KUKA KRL program: vw_mod_usr_r.src, vw_mod_usr_r.dat

--- vw_mod_usr_r.src ---
&ACCESS RV2
&REL 1
&COMMENT KS26
&PARAM TPUSER_VERSION = 8.3.0
&PARAM DISKPATH = KRC:\R1\VW_User\Applikation\Projekt_Modul
DEF VW_MOD_USR_R( )
;
;***************************************************
;*Technologiepaket Projekt Modul                   *
;*                                                 *
;*Konzernstandard                                  *
;*Bearbeiter: C. Eisenknappl AUDI AG I/PG-C61      *
;*                                                 *
;* Erstellt am:                                    *
;*                                                 *
;***************************************************
;
END
;
;FOLD MOD1_Interface
GLOBAL DEF MOD1_Interface(USER_CMD:IN,CMD_SEL:IN,PAR1:IN,PAR2:IN,PAR3:IN,PAR4:IN,PAR5:IN,PAR6:IN,PAR7:IN,PAR8:IN,PAR9:IN)
DECL VW_USER_CMD USER_CMD
INT  CMD_SEL,PAR1,PAR2,PAR3,PAR4,PAR5,PAR6,PAR7,PAR8,PAR9
INT i
BOOL bRet
;
SWITCH USER_CMD
;
;***************************************************
  CASE #USR_INIT
    ;FOLD Init
    ;
    ;
    ;ENDFOLD (Init)
;
;***************************************************
  CASE #USR_ADV
    ;FOLD Advance
    ;
    ;
    ;ENDFOLD (Advance)
;
;***************************************************
  CASE #USR_TRIG
    ;FOLD Trig
    ;
    ;
    ;ENDFOLD (TRIG)
;
;***************************************************
  CASE #USR_MAIN
    ;FOLD Main
    ;
    ;
    ;ENDFOLD (Main)
;
;***************************************************
  CASE #USR_MAKRO
    ;FOLD MAKRO
    ;
    ;
    ;ENDFOLD (Makro)
    ;
;***************************************************
ENDSWITCH ;(USER_CMD)
END
;
;ENDFOLD (MOD1_Interface)
;
;***************************************************
;FOLD MOD1 Zangenfunktion
;
;
;ENDFOLD (Zangenfunktion)
;
;***************************************************
;FOLD MOD1_Meldungen
DEF MOD1_Msg(msg_nr :IN, MsgTyp :IN)
INT msg_nr
DECL MOD1R_MsgType MsgTyp
DECL KrlMsg_T USER_MSG
DECL KrlMsgPar_T Par[3]
DECL KrlMsgOpt_T Opt
DECL STATE_T Stat
;
USER_MSG={ Modul[] "MOD1_R_Msg", Nr -1, Msg_txt[] " "}
Opt={ VL_Stop TRUE, Clear_P_Reset TRUE, Log_To_DB FALSE }
Par[1]={ Par_type #Value, Par_txt[] " " }
;
IF ((n_MOD1R_Handle[msg_nr]<0) OR (MsgTyp==#NotifyMsg) OR (MsgTyp==#QuitMsg)) THEN
  USER_MSG.Nr=msg_nr
  SWITCH msg_nr
    CASE 1
      USER_MSG.MSG_TXT[]=" "
    CASE 2
      USER_MSG.MSG_TXT[]=" "
    CASE 3
      USER_MSG.MSG_TXT[]=" "
    CASE 4
      USER_MSG.MSG_TXT[]=" "
    CASE 5
      USER_MSG.MSG_TXT[]=" "
    CASE 6
      USER_MSG.MSG_TXT[]=" "
    CASE 7
      USER_MSG.MSG_TXT[]=" "
    CASE 8
      USER_MSG.MSG_TXT[]=" "
    CASE 9
      USER_MSG.MSG_TXT[]=" "
    CASE 10
      USER_MSG.MSG_TXT[]=" "
    DEFAULT
      USER_MSG.MSG_TXT[]="unbekannte Meldung"
  ENDSWITCH
  SWITCH MsgTyp
    CASE #StateMsg
      n_MOD1R_Handle[msg_nr]=Set_KrlMsg (#State, USER_MSG, Par[], Opt) ;Ausgabe Statusmeldung
    CASE #QuitMsg
      n_MOD1R_Handle[msg_nr]=Set_KrlMsg (#Quit, USER_MSG, Par[], Opt) ;Ausgabe Quittierungsmeldung
      WHILE (Exists_KrlMsg(n_MOD1R_Handle[msg_nr]))  ;Warten bis der Anwender quittiert
        WAIT SEC 0.1
      ENDWHILE
    CASE #NotifyMsg
      n_MOD1R_Handle[msg_nr]=Set_KrlMsg (#Notify, USER_MSG, Par[], Opt) ;Ausgabe Hinweismeldung
    DEFAULT
      n_MOD1R_Handle[msg_nr]=Set_KrlMsg (#Quit, USER_MSG, Par[], Opt) ;Ausgabe Quittierungsmeldung
  ENDSWITCH
ENDIF
END
;
;ENDFOLD (MOD1 Meldungen)
;
;***************************************************
;FOLD MOD2_Interface
GLOBAL DEF MOD2_Interface(USER_CMD:IN,CMD_SEL:IN,PAR1:IN,PAR2:IN,PAR3:IN,PAR4:IN,PAR5:IN,PAR6:IN,PAR7:IN,PAR8:IN,PAR9:IN)
DECL VW_USER_CMD USER_CMD
INT  CMD_SEL,PAR1,PAR2,PAR3,PAR4,PAR5,PAR6,PAR7,PAR8,PAR9
INT i
BOOL bRet
;
SWITCH USER_CMD
;
;***************************************************
  CASE #USR_INIT
    ;FOLD Init
    ;
    $OUT[O_BT_FEHL] = FALSE
    $FLAG[F_X_Lauf_nio] = FALSE
    $FLAG[F_Y_Lauf_nio] = FALSE
    $FLAG[F_Z_Lauf_nio] = FALSE
    $FLAG[F_XYZ_OutOfRange] = FALSE
    VisuKorrWert=$NULLFRAME
    ;
    ;ENDFOLD (Init)
;
;***************************************************
  CASE #USR_ADV
    ;FOLD Advance
    ;
    SWITCH PAR1
      CASE 1 ; VW_xyz-Scan

    DEFAULT
      ;
    ENDSWITCH
    ;
    ;ENDFOLD (Advance)
;
;***************************************************
  CASE #USR_TRIG
    ;FOLD Trig
    ;
    SWITCH PAR1
      CASE 1 ; VW_xyz-Scan

    DEFAULT
      ;
    ENDSWITCH
    ;
    ;ENDFOLD (TRIG)
;
;***************************************************
  CASE #USR_MAIN
    ;FOLD Main
    ;
    SWITCH PAR1
      CASE 1 ; VW_xyz-Scan
        XYZ_MODE=1 ; Art der MESSUNG, 1: x,y,z, sonst: scan_Circ (not supported)
        XYZ_Fct=PAR2 ; Funktion, 21: Messfahrt, 22:Referenzfahrt, 23:Nullsetzen, 24: Berechnung Korrektur
        XYZ_Rtng=PAR3 ; Such-Richtung, Par3=1+n*3: x, Par3=2+n*3: y, Par3=3+n*3: z
        XYZ_BaseNr=PAR4; Base-Nr mit der MESSUNG durchgefuehrt wird
        XYZ_Suchweg=PAR5 ; Suchstrecke in [mm]
        XYZ_C_Mess=PAR6 ; Nummer Starteingang fuer Interrupt
        ;
        ;Funktion VW-XYZ-Scan (Init,Ref,Messen,Calc)
        WHILE (XYZ_Rtng<21) OR (XYZ_Rtng>44) ; selection out of range
          MOD2_Msg(33, #QuitMsg) ;Falsche Richtung PAR3
          RETURN
        ENDWHILE
        ;Check act. Base-Nr
        WHILE ((VW_MPARA_ACT.BASE_NO<1) OR (VW_MPARA_ACT.BASE_NO>32)) AND (XYZ_Fct <> 21) ; selection out of range
          MOD2_Msg(42, #QuitMsg) ;Base-Nr ungueltig
          RETURN
        ENDWHILE
        SWITCH XYZ_Rtng
          CASE 21, 24, 27, 30, 33, 36, 39, 42 ; Gruppe X
            MODELL=(XYZ_Rtng-18)/3
          CASE 22, 25, 28, 31, 34, 37, 40, 43 ; Gruppe Y
            MODELL=(XYZ_Rtng-19)/3
          CASE 23, 26, 29, 32, 35, 38, 41, 44 ; Gruppe Z
            MODELL=(XYZ_Rtng-20)/3
          DEFAULT
            MOD2_Msg(33, #QuitMsg) ;Richtung ungueltig
            HALT
        ENDSWITCH
        $OUT[O_BT_FEHL] = FALSE
        $FLAG[F_X_Lauf_nio] = FALSE
        $FLAG[F_Y_Lauf_nio] = FALSE
        $FLAG[F_Z_Lauf_nio] = FALSE
        $FLAG[F_XYZ_OutOfRange] = FALSE
        VisuKorrWert=$NULLFRAME
        SWITCH XYZ_Fct
          CASE 21 ; Base auf $nullframe setzen
            Base_init()
          CASE 22 ; Funktion Ref-Fahrt
            WHILE ($CYCFLAG[XYZ_C_Mess]== FALSE)
              MOD2_Msg(40, #StateMsg) ;Suchlaufsensor defekt!
              HALT
            ENDWHILE
            scan_xyz()
            IF NOT MESSUNG THEN
              MOD2_Msg(41, #StateMsg) ;Interrupt nicht geschaltet!
              HALT
            ENDIF
          CASE 23 ; Funktion Messfahrt
            WHILE ($CYCFLAG[XYZ_C_Mess]== FALSE)
              MOD2_Msg(40, #StateMsg) ;Suchlaufsensor defekt!
              HALT
            ENDWHILE
            scan_xyz()
            IF (MESSUNG AND NOT $FLAG[F_XYZ_OutOfRange]) THEN
              BASE_BERECHNUNG()
            ELSE
              $OUT[O_BT_FEHL] = TRUE
              MOD2_Msg(39, #StateMsg) ;Roboter faehrt ohne Korrektur!
              HALT
            ENDIF
          DEFAULT
            MOD2_Msg(32, #QuitMsg) ;Falsche Funktion PAR2
        ENDSWITCH
      DEFAULT
        ;
    ENDSWITCH
    ;
    ;ENDFOLD (Main)
;
;***************************************************
  CASE #USR_MAKRO
    ;FOLD MAKRO
    ;
    ;
    ;ENDFOLD (Makro)
    ;
;***************************************************
ENDSWITCH ;(USER_CMD)
END
;
;ENDFOLD (MOD2_Interface)
;
;***************************************************
;FOLD MOD2 Zangenfunktion
;
;
;ENDFOLD (Zangenfunktion)
;
;***************************************************
;FOLD MOD2_Meldungen
DEF MOD2_Msg(msg_nr :IN, MsgTyp :IN)
INT msg_nr, Hilfsint
DECL MOD2R_MsgType MsgTyp
DECL KrlMsg_T USER_MSG
DECL KrlMsgPar_T Par[3]
DECL KrlMsgOpt_T Opt
DECL STATE_T Stat
REAL HilfsReal
;
USER_MSG = { Modul[] "MOD2_R_Msg", Nr -1, Msg_txt[] " "}
Opt = { VL_Stop True, Clear_P_Reset True, Log_To_DB False }
Par[1] = { Par_type #Value, Par_txt[] " " }
;
IF ((n_MOD2R_Handle[msg_nr]<0) OR (MsgTyp==#NotifyMsg) OR (MsgTyp==#QuitMsg)) THEN
  USER_MSG.Nr = msg_nr
  SWITCH msg_nr
    CASE 11
      USER_MSG.MSG_TXT[]="Base wurde initialisiert."
    CASE 12
      USER_MSG.MSG_TXT[]="Ref-Pos wurde gespeichert."
    CASE 13
      USER_MSG.MSG_TXT[]="Mess-Pos wurde gespeichert."
    CASE 14
      Par[1] = { Par_type #Value, par_real 1}
      ;Real auf zwei Nachkommastellen runden
      HilfsReal = VisuKorrWert.x*100
      HilfsInt = HilfsReal*1
      Par[1].par_real = HilfsInt*0.01
      Par[2] = { Par_type #Value, par_real 1}
      ;Real auf zwei Nachkommastellen runden
      HilfsReal = VisuKorrWert.y*100
      HilfsInt = HilfsReal*1
      Par[2].par_real = HilfsInt*0.01
      Par[3] = { Par_type #Value, par_real 1}
      ;Real auf zwei Nachkommastellen runden
      HilfsReal = VisuKorrWert.z*100
      HilfsInt = HilfsReal*1
      Par[3].par_real = HilfsInt*0.01
      USER_MSG.MSG_TXT[]="Basedaten berechnet. Korrekturen [mm]: x %1,y %2, z %3"
    CASE 31
      USER_MSG.MSG_TXT[]="Falsche Messart PAR1"
    CASE 32
      USER_MSG.MSG_TXT[]="Falsche Funktion PAR2"
    CASE 33
      USER_MSG.MSG_TXT[]="Falsche Richtung PAR3"
    CASE 34
      USER_MSG.MSG_TXT[]="Meldung nicht Deklariert"
    CASE 35
      USER_MSG.MSG_TXT[]="Falsche Bezugsbase PAR5"
    CASE 36
      USER_MSG.MSG_TXT[]="MESSUNG in X fehlerhaft"
    CASE 37
      USER_MSG.MSG_TXT[]="MESSUNG in Y fehlerhaft"
    CASE 38
      USER_MSG.MSG_TXT[]="MESSUNG in Z fehlerhaft"
    CASE 39
      USER_MSG.MSG_TXT[]="Roboter faehrt ohne Korrektur!"
    CASE 40
      USER_MSG.MSG_TXT[]="Suchlaufsensor defekt!"
    CASE 41
      USER_MSG.MSG_TXT[]="Interrupt nicht geschaltet! Sensor defekt?"
    CASE 42
      USER_MSG.MSG_TXT[]="Aktuelle Base-Nummer ungueltig!"
    CASE 51
      USER_MSG.MSG_TXT[]="Par 1 falscher Wert!"
    DEFAULT
      USER_MSG.MSG_TXT[]="unbekannte Meldung"
  ENDSWITCH
  SWITCH MsgTyp
    CASE #StateMsg
      n_MOD2R_Handle[msg_nr] = Set_KrlMsg (#State, USER_MSG, Par[], Opt) ;Ausgabe Statusmeldung
    CASE #QuitMsg
      n_MOD2R_Handle[msg_nr] = Set_KrlMsg (#Quit, USER_MSG, Par[], Opt) ;Ausgabe Quittierungsmeldung
      While ( Exists_KrlMsg(n_MOD2R_Handle[msg_nr]) )  ;Warten bis der Anwender quittiert
        Wait Sec 0.1
      Endwhile
    CASE #NotifyMsg
      n_MOD2R_Handle[msg_nr] = Set_KrlMsg (#Notify, USER_MSG, Par[], Opt) ;Ausgabe Hinweismeldung
    DEFAULT
      n_MOD2R_Handle[msg_nr] = Set_KrlMsg (#Quit, USER_MSG, Par[], Opt) ;Ausgabe Quittierungsmeldung
  ENDSWITCH
ENDIF
END
;
;ENDFOLD (MOD2 Meldungen)
;
;***************************************************
;FOLD MOD3_Interface
GLOBAL DEF MOD3_Interface(USER_CMD:IN,CMD_SEL:IN,PAR1:IN,PAR2:IN,PAR3:IN,PAR4:IN,PAR5:IN,PAR6:IN,PAR7:IN,PAR8:IN,PAR9:IN)
DECL VW_USER_CMD USER_CMD
INT  CMD_SEL,PAR1,PAR2,PAR3,PAR4,PAR5,PAR6,PAR7,PAR8,PAR9
INT i
BOOL bRet
;
SWITCH USER_CMD
;
;***************************************************
  CASE #USR_INIT
    ;FOLD Init
    ;
    ;
    ;ENDFOLD (Init)
;
;***************************************************
  CASE #USR_ADV
    ;FOLD Advance
    ;
    ;
    ;ENDFOLD (Advance)
;
;***************************************************
  CASE #USR_TRIG
    ;FOLD Trig
    ;
    ;
    ;ENDFOLD (TRIG)
;
;***************************************************
  CASE #USR_MAIN
    ;FOLD Main
    ;
    ;
    ;ENDFOLD (Main)
;
;***************************************************
  CASE #USR_MAKRO
    ;FOLD MAKRO
    ;
    ;
    ;ENDFOLD (Makro)
    ;
;***************************************************
ENDSWITCH ;(USER_CMD)
END
;
;ENDFOLD (MOD3_Interface)
;
;***************************************************
;FOLD MOD3 Zangenfunktion
;
;
;ENDFOLD (Zangenfunktion)
;
;***************************************************
;FOLD MOD3_Meldungen
DEF MOD3_Msg(msg_nr :IN, MsgTyp :IN)
INT msg_nr
DECL MOD1R_MsgType MsgTyp
DECL KrlMsg_T USER_MSG
DECL KrlMsgPar_T Par[3]
DECL KrlMsgOpt_T Opt
DECL STATE_T Stat
;
USER_MSG={ Modul[] "MOD3_R_Msg", Nr -1, Msg_txt[] " "}
Opt={ VL_Stop TRUE, Clear_P_Reset TRUE, Log_To_DB FALSE }
Par[1]={ Par_type #Value, Par_txt[] " " }
;
IF ((n_MOD3R_Handle[msg_nr]<0) OR (MsgTyp==#NotifyMsg) OR (MsgTyp==#QuitMsg)) THEN
  USER_MSG.Nr=msg_nr
  SWITCH msg_nr
    CASE 1
      USER_MSG.MSG_TXT[]=" "
    CASE 2
     USER_MSG.MSG_TXT[]=" "
    CASE 3
      USER_MSG.MSG_TXT[]=" "
    CASE 4
      USER_MSG.MSG_TXT[]=" "
    CASE 5
      USER_MSG.MSG_TXT[]=" "
    CASE 6
      USER_MSG.MSG_TXT[]=" "
    CASE 7
      USER_MSG.MSG_TXT[]=" "
    CASE 8
      USER_MSG.MSG_TXT[]=" "
    CASE 9
      USER_MSG.MSG_TXT[]=" "
    CASE 10
      USER_MSG.MSG_TXT[]=" "
    DEFAULT
      USER_MSG.MSG_TXT[]="unbekannte Meldung"
  ENDSWITCH
  SWITCH MsgTyp
    CASE #StateMsg
      n_MOD3R_Handle[msg_nr]=Set_KrlMsg (#State, USER_MSG, Par[], Opt) ;Ausgabe Statusmeldung
    CASE #QuitMsg
      n_MOD3R_Handle[msg_nr]=Set_KrlMsg (#Quit, USER_MSG, Par[], Opt) ;Ausgabe Quittierungsmeldung
      WHILE (Exists_KrlMsg(n_MOD3R_Handle[msg_nr]))  ;Warten bis der Anwender quittiert
        WAIT SEC 0.1
      ENDWHILE
    CASE #NotifyMsg
      n_MOD3R_Handle[msg_nr]=Set_KrlMsg (#Notify, USER_MSG, Par[], Opt) ;Ausgabe Hinweismeldung
    DEFAULT
      n_MOD3R_Handle[msg_nr]=Set_KrlMsg (#Quit, USER_MSG, Par[], Opt) ;Ausgabe Quittierungsmeldung
  ENDSWITCH
ENDIF
END
;
;ENDFOLD (MOD3 Meldungen)
;
;***************************************************
;FOLD DZ Interface
GLOBAL DEF DZ_Interface(USER_CMD:IN,CMD_SEL:IN,PAR1:IN,PAR2:IN,PAR3:IN,PAR4:IN,PAR5:IN,PAR6:IN,PAR7:IN,PAR8:IN,PAR9:IN)
DECL VW_USER_CMD USER_CMD
INT CMD_SEL,PAR1,PAR2,PAR3,PAR4,PAR5,PAR6,PAR7,PAR8,PAR9
INT i
;
;***************************************************
SWITCH USER_CMD
;
;***************************************************
  CASE #USR_INIT
    ;FOLD Init
    ;
    ;
    ;ENDFOLD (Init)
;
;***************************************************
  CASE #USR_ADV
    ;FOLD Advance
    ;
    ;
    ;ENDFOLD (Advance)
;
;***************************************************
  CASE #USR_TRIG
    ;FOLD Trig
    ;
    ;
    ;ENDFOLD (Trig)
;
;***************************************************
  CASE #USR_MAIN
    ;FOLD Main
    ;
    ;
    ;ENDFOLD (Main)
;
;***************************************************
  CASE #USR_MAKRO
    ;FOLD Makro
    ;
    SWITCH PAR1
      CASE 21 ; Handling
        SWITCH PAR2
          CASE 2101, 2102  ;Setze Ansteuerung
            DZ_busy=TRUE
            DZ_fm=FALSE
            FOR i = 1 TO AnzSpnGr
              IF ($FLAG[i]==TRUE) THEN
                dzSpnGrYr[i]=PAR2-2100
              ENDIF
            ENDFOR
            DZ_busy=FALSE
          CASE 2103  ;Setze Stellung
            DZ_busy=TRUE
            FOR i = 1 TO AnzSpnGr
              IF (i<17) THEN ;zwei Positionen
                IF ($CYCFLAG[30+i]==FALSE) AND  ($CYCFLAG[30+(i*2)]==TRUE) THEN
                  dzSpnGrKe[i]=1
                ENDIF
                IF ($CYCFLAG[30+i]==TRUE) AND  ($CYCFLAG[30+(i*2)]==FALSE) THEN
                  dzSpnGrKe[i]=2
                ENDIF
              ELSE ;eine Position
                IF ($CYCFLAG[30+i]==TRUE) THEN
                  dzSpnGrKe[i]=1
                ELSE
                  dzSpnGrKe[i]=2
                ENDIF
              ENDIF
            ENDFOR
            DZ_fm=TRUE
            DZ_busy=FALSE
          CASE 2104  ;Auswertung
            DZ_busy=TRUE

            DZ_busy=FALSE
          DEFAULT
            ;
        ENDSWITCH
      DEFAULT
        ;
    ENDSWITCH
    ;
    ;ENDFOLD (Makro)
;
;***************************************************
  DEFAULT
;
  ENDSWITCH
END
;
;ENDFOLD (DZ Interface)
;
;***************************************************
;FOLD Subroutinen
;***************************************************
;FOLD scan_xyz
DEF scan_xyz()

  START_POS=$NULLFRAME
  ;
  ;Interrupts initialisieren
  INTERRUPT DECL 15 WHEN NOT $CYCFLAG[XYZ_C_Mess] DO TCP_MESS1 ()
  MESSUNG = FALSE
  OV_MERK=$OV_PRO
  $OV_PRO=XYZ_vRED
  ;Startpunkt fuer den Messlauf anfahren
  LIN  $POS_ACT
  START_POS=$pos_act
  INTERRUPT ON 15
  ;Suchbewegung
  SUCH_MOVE()
  ;Interrupts ausschalten
  INTERRUPT OFF 15
  $OV_PRO=OV_MERK
  $ADVANCE=1
  LIN START_POS
  ;
  IF MESSUNG_X OR MESSUNG_Y OR MESSUNG_Z THEN
    IF (MESSUNG_X AND MESSUNG_Y) OR (MESSUNG_X AND MESSUNG_Z) OR (MESSUNG_Y AND MESSUNG_Z) THEN
      SWITCH XYZ_Rtng
        CASE 21,24,27,30,33,36,39,42
          $FLAG[F_X_Lauf_nio] = TRUE
          IF(MESSUNG_X== FALSE) THEN
            MOD2_Msg(36, #NotifyMsg) ;MESSUNG in X fehlerhaft
          ENDIF
        CASE 22,25,28,31,34,37,40,43
          $FLAG[F_Y_Lauf_nio] = TRUE
          IF(MESSUNG_Y== FALSE) THEN
            MOD2_Msg(37, #NotifyMsg) ;MESSUNG in Y fehlerhaft
          ENDIF
        CASE 23,26,29,32,35,38,41,44
          $FLAG[F_Z_Lauf_nio] = TRUE
          IF(MESSUNG_Z== FALSE) THEN
            MOD2_Msg(38, #NotifyMsg) ;MESSUNG in Z fehlerhaft
          ENDIF
        DEFAULT
          MOD2_Msg(33, #QuitMsg) ;Falsche Richtung PAR3
      ENDSWITCH
    ELSE
      MESSUNG=MESSUNG_X OR MESSUNG_Y OR MESSUNG_Z
    ENDIF
  ELSE
    $FLAG[F_XYZ_OutOfRange] = TRUE
  ENDIF
  ;
END
;ENDFOLD scan_xyz
;
;***************************************************
;FOLD BASE_BERECHNUNG
DEF BASE_BERECHNUNG()

  INT OFFSET
  DECL STATE_T STATE
  BOOL hilf

  hilf = FALSE
  IF(XYZ_BaseNr<21) OR (XYZ_BaseNr>31) THEN
    MOD2_Msg(35, #QuitMsg) ;Falsche Bezugsbase PAR5
  ELSE
    korr_wert=$NULLFRAME
    SWITCH XYZ_Rtng
      CASE 21,24,27,30,33,36,39,42
        IF(MESSUNG_X== TRUE) THEN
          korr_wert.x=XYZ_MESS_POS[MODELL,1].x-XYZ_REF_POS[MODELL,1].x
          hilf = TRUE
        ENDIF
      CASE 22,25,28,31,34,37,40,43
        IF(MESSUNG_Y== TRUE) THEN
          korr_wert.y=XYZ_MESS_POS[MODELL,2].y-XYZ_REF_POS[MODELL,2].y
          hilf = TRUE
        ENDIF
      CASE 23,26,29,32,35,38,41,44
        IF(MESSUNG_Z== TRUE) THEN
          korr_wert.z=XYZ_MESS_POS[MODELL,3].z-XYZ_REF_POS[MODELL,3].z
          hilf = TRUE
        ENDIF
      DEFAULT
        MOD2_Msg(33, #QuitMsg) ;Falsche Richtung PAR3
    ENDSWITCH

    IF(hilf== TRUE) THEN
      XyzBaseOld=base_data[XYZ_BaseNr]
      base_data[XYZ_BaseNr]=base_data[XYZ_BaseNr]:korr_wert
      VisuKorrWert=$NULLFRAME
      VisuKorrWert.X=base_data[XYZ_BaseNr].X-XyzBaseOld.X
      VisuKorrWert.Y=base_data[XYZ_BaseNr].Y-XyzBaseOld.Y
      VisuKorrWert.Z=base_data[XYZ_BaseNr].Z-XyzBaseOld.Z
      IF($MODE_OP <> #EX) OR (XYZ_KORR_DBG == TRUE) THEN
        MOD2_Msg(14, #NotifyMsg) ;Basedaten berechnet
      ENDIF
      datum=$date
      offset=0
      swrite(korr_tab[log_nr].korr_wert[],state,offset,"x: %.2f,y: %.2f, z: %.2f",korr_wert.x,korr_wert.y,korr_wert.z)
      offset=0
      swrite(korr_tab[log_nr].korr_datum[],state,offset,"%d.%d.%d  %d:%d:%d",datum.day,datum.month,datum.year,datum.hour,datum.min,datum.sec)
      log_nr=log_nr+1
      IF log_nr>50 THEN
        log_nr=1
      ENDIF
    ELSE
      korr_wert=$nullframe
      datum=$date
      offset=0
      swrite(korr_tab[log_nr].korr_wert[],state,offset,"x: %.2f,y: %.2f, z: %.2f",korr_wert.x,korr_wert.y,korr_wert.z)
      offset=0
      swrite(korr_tab[log_nr].korr_datum[],state,offset,"%d.%d.%d  %d:%d:%d",datum.day,datum.month,datum.year,datum.hour,datum.min,datum.sec)
      log_nr=log_nr+1
      IF log_nr>50 THEN
        log_nr=1
      ENDIF
      MOD2_Msg(39, #StateMsg) ;Roboter faehrt ohne Korrektur!
    ENDIF
  ENDIF
END
;ENDFOLD BASE_BERECHNUNG
;
;***************************************************
;FOLD SUCH_MOVE
DEF SUCH_MOVE ()

  FRAME LIN_ZIEL
  FRAME SUCH_STRECKE

  SUCH_STRECKE=$nullframe
  MESSUNG_X = FALSE
  MESSUNG_Y = FALSE
  MESSUNG_Z = FALSE

  SWITCH XYZ_Rtng
    CASE 21,24,27,30,33,36,39,42
      SUCH_STRECKE.x=-XYZ_Suchweg
      LIN_REL SUCH_STRECKE
    CASE 22,25,28,31,34,37,40,43
      SUCH_STRECKE.y=-XYZ_Suchweg
      LIN_REL SUCH_STRECKE
    CASE 23,26,29,32,35,38,41,44
      SUCH_STRECKE.z=-XYZ_Suchweg
      LIN_REL SUCH_STRECKE
    DEFAULT
      MOD2_Msg(33, #NotifyMsg) ;Falsche Richtung PAR3
  ENDSWITCH
  $ADVANCE=0
END
;ENDFOLD SUCH_MOVE
;
;***************************************************
;FOLD TCP_MESS1
DEF TCP_MESS1 ()
  SWITCH XYZ_Fct
    CASE 22
      BASE_ORG=BASE_DATA[VW_MPARA_ACT.BASE_NO]
      SWITCH XYZ_Rtng
        CASE 21,24,27,30,33,36,39,42
          XYZ_REF_POS[MODELL,1]=$POS_INT
        CASE 22,25,28,31,34,37,40,43
          XYZ_REF_POS[MODELL,2]=$POS_INT
        CASE 23,26,29,32,35,38,41,44
          XYZ_REF_POS[MODELL,3]=$POS_INT
        DEFAULT
      ENDSWITCH
      IF($MODE_OP <> #EX) THEN
        MOD2_Msg(12, #StateMsg) ;Ref-Pos wurde gespeichert
      ENDIF
      BRAKE
    CASE 23
      SWITCH XYZ_Rtng
        CASE 21,24,27,30,33,36,39,42
          XYZ_MESS_POS[MODELL,1]=$POS_INT
          MESSUNG_X = TRUE
        CASE 22,25,28,31,34,37,40,43
          XYZ_MESS_POS[MODELL,2]=$POS_INT
          MESSUNG_Y = TRUE
        CASE 23,26,29,32,35,38,41,44
          XYZ_MESS_POS[MODELL,3]=$POS_INT
          MESSUNG_Z = TRUE
        DEFAULT
      ENDSWITCH
      IF($MODE_OP <> #EX) AND (MESSUNG_X OR MESSUNG_Y OR MESSUNG_Z) THEN
		MOD2_Msg(13, #NotifyMsg) ;Mess-Pos wurde gespeichert.
      ENDIF
      BRAKE
    DEFAULT
      HALT
      MOD2_Msg(32, #QuitMsg) ;Falsche Funktion PAR2
  ENDSWITCH

  SWITCH XYZ_Rtng
    CASE 21,24,27,30,33,36,39,42
      MESSUNG_X = TRUE
    CASE 22,25,28,31,34,37,40,43
      MESSUNG_Y = TRUE
    CASE 23,26,29,32,35,38,41,44
      MESSUNG_Z = TRUE
    DEFAULT
      MOD2_Msg(33, #QuitMsg) ;Falsche Richtung PAR3
  ENDSWITCH
  RESUME

END
;ENDFOLD BASE_BERECHNUNG
;
;***************************************************
;FOLD BASE_INIT
DEF BASE_INIT()
  IF(XYZ_BaseNr<21) OR (XYZ_BaseNr>31) THEN
    MOD2_Msg(35, #QuitMsg) ;Falsche Bezugsbase PAR5
  ELSE
    BASE_DATA[XYZ_BaseNr]=BASE_ORG
    IF($MODE_OP <> #EX) THEN
      MOD2_Msg(11, #NotifyMsg) ;Base wurde initialisiert.
    ENDIF
  ENDIF
END
;ENDFOLD BASE_INIT
;
;***************************************************
;FOLD DZ LogBaseCorr
;
GLOBAL DEF DZ_LogBaseCorr(sender :IN, corrType :IN, corrFrame :IN, baseNr :IN)
;
DECL CHAR sender[] ;should be name of calling user-module (Bsp. vw_xml_usr)
DECL CHAR corrType[] ;only abs, rel
DECL FRAME corrFrame
DECL STATE_T state
DECL DATE DATUM
INT baseNr

;DZ_LogBaseCorr(vw_xyz_usr_r,abs,BASE_DATA[3],3)

DATUM=$date
offset=0
swrite(dzCorrTab[logNr].dzSender[],state,offset,"                ")
offset=0
swrite(dzCorrTab[logNr].dzSender[],state,offset,"%s",sender[])
;
offset=0
swrite(dzCorrTab[logNr].dzCorrType[],state,offset,"   ")
offset=0
swrite(dzCorrTab[logNr].dzCorrType[],state,offset,"%s",corrType[])
;
offset=0
swrite(dzCorrTab[logNr].dzCorr[],state,offset,"    ")
offset=0
On_Error_Proceed
swrite(dzCorrTab[logNr].dzCorr[],state,offset,"x %.1f y %.1f z %.1f a %.4f b %.4f c %.4f",corrFrame.x,corrFrame.y,corrFrame.z,corrFrame.a,corrFrame.b,corrFrame.c)
;
offset=0
swrite(dzCorrTab[logNr].dzCorrBase[],state,offset,"  ")
offset=0
swrite(dzCorrTab[logNr].dzCorrBase[],state,offset,"%d",baseNr)
;
offset=0
swrite(dzCorrTab[logNr].dzLogDatum[],state,offset,"%d.%d.%d  %d:%d:%d",datum.day,datum.month,datum.year,datum.hour,datum.min,datum.sec)
;
logNr=logNr+1
IF logNr>200 then
  logNr=1
ENDIF
;
END
;
;ENDFOLD (DZ_LogBaseCorr)
;***************************************************
;ENDFOLD (Subroutinen)
;

--- vw_mod_usr_r.dat ---
&ACCESS  RV
&COMMENT KS26
&PARAM DISKPATH = VW_User/Applikation/Projekt_Modul
&PARAM TPUSER_VERSION = 8.3.0
&REL 1
DEFDAT  vw_mod_usr_r PUBLIC
;
;***************************************************
;*Technologiepaket Projekt_Modul                   *
;*                                                 *
;*Konzernstandard                                  *
;*Bearbeiter: C. Eisenknappl AUDI AG I/PG-C61      *
;*                                                 *
;* Erstellt am:                                    *
;*                                                 *
;***************************************************
;
;FOLD MOD1
;
;
;***************************************************
;FOLD Meldungsausgabe
ENUM MOD1R_MsgType StateMsg,QuitMsg,NotifyMsg
;ENDFOLD
;***************************************************
;ENDFOLD (MOD1)
;
;***************************************************
;FOLD MOD2
;
;FOLD VW_xyz-Scan
;
;FOLD INTEGER
INT XYZ_MODE=0
INT XYZ_Fct=22
INT XYZ_Rtng=44
INT XYZ_BaseNr=21
INT XYZ_C_Mess=1
INT XYZ_Suchweg=5
INT ov_merk=30
INT F_X_Lauf_nio=785
INT F_Y_Lauf_nio=786
INT F_Z_Lauf_nio=787
INT F_XYZ_OutOfRange=788
INT O_BT_FEHL=123
INT MODELL=1
INT FUNKTION,RICHTUNG,STRECKE,WZG_NR,EINGANG
INT LOG_NR=1
GLOBAL INT XYZ_vRED=6 ;PrgOv waehrend Suchfahrt in %
;ENDFOLD INTEGER
;
;FOLD BOOLEAN
BOOL MESSUNG
BOOL MESSUNG_X=FALSE
BOOL MESSUNG_Y=TRUE
BOOL MESSUNG_Z=FALSE
GLOBAL BOOL XYZ_KORR_DBG=FALSE ;Korrekturwerte anzeigen/nicht anzeigen
;ENDFOLD BOOLEAN
;
;FOLD FRAMES
FRAME START_POS={X 0.0,Y 0.0,Z 0.0,A 0.0,B 0.0,C 0.0}
FRAME KORR_WERT={X 0.0,Y 0.0,Z 0.0,A 0.0,B 0.0,C 0.0}
FRAME BASE_ORG={X 0.0,Y 0.0,Z 0.0,A 0.0,B 0.0,C 0.0}
FRAME VisuKorrWert={X 0.0,Y 0.0,Z 0.0,A 0.0,B 0.0,C 0.0}
FRAME XyzBaseOld={X 0.0,Y 0.0,Z 0.0,A 0.0,B 0.0,C 0.0}
;
GLOBAL FRAME XYZ_MESS_POS[8,3]
XYZ_MESS_POS[1,1]={X 0.0,Y 0.0,Z 0.0,A 0.0,B 0.0,C 0.0}
XYZ_MESS_POS[1,2]={X 0.0,Y 0.0,Z 0.0,A 0.0,B 0.0,C 0.0}
XYZ_MESS_POS[1,3]={X 0.0,Y 0.0,Z 0.0,A 0.0,B 0.0,C 0.0}
XYZ_MESS_POS[2,1]={X 0.0,Y 0.0,Z 0.0,A 0.0,B 0.0,C 0.0}
XYZ_MESS_POS[2,2]={X 0.0,Y 0.0,Z 0.0,A 0.0,B 0.0,C 0.0}
XYZ_MESS_POS[2,3]={X 0.0,Y 0.0,Z 0.0,A 0.0,B 0.0,C 0.0}
XYZ_MESS_POS[3,1]={X 0.0,Y 0.0,Z 0.0,A 0.0,B 0.0,C 0.0}
XYZ_MESS_POS[3,2]={X 0.0,Y 0.0,Z 0.0,A 0.0,B 0.0,C 0.0}
XYZ_MESS_POS[3,3]={X 0.0,Y 0.0,Z 0.0,A 0.0,B 0.0,C 0.0}
XYZ_MESS_POS[4,1]={X 0.0,Y 0.0,Z 0.0,A 0.0,B 0.0,C 0.0}
XYZ_MESS_POS[4,2]={X 0.0,Y 0.0,Z 0.0,A 0.0,B 0.0,C 0.0}
XYZ_MESS_POS[4,3]={X 0.0,Y 0.0,Z 0.0,A 0.0,B 0.0,C 0.0}
XYZ_MESS_POS[5,1]={X 0.0,Y 0.0,Z 0.0,A 0.0,B 0.0,C 0.0}
XYZ_MESS_POS[5,2]={X 0.0,Y 0.0,Z 0.0,A 0.0,B 0.0,C 0.0}
XYZ_MESS_POS[5,3]={X 0.0,Y 0.0,Z 0.0,A 0.0,B 0.0,C 0.0}
XYZ_MESS_POS[6,1]={X 0.0,Y 0.0,Z 0.0,A 0.0,B 0.0,C 0.0}
XYZ_MESS_POS[6,2]={X 0.0,Y 0.0,Z 0.0,A 0.0,B 0.0,C 0.0}
XYZ_MESS_POS[6,3]={X 0.0,Y 0.0,Z 0.0,A 0.0,B 0.0,C 0.0}
XYZ_MESS_POS[7,1]={X 0.0,Y 0.0,Z 0.0,A 0.0,B 0.0,C 0.0}
XYZ_MESS_POS[7,2]={X 0.0,Y 0.0,Z 0.0,A 0.0,B 0.0,C 0.0}
XYZ_MESS_POS[7,3]={X 0.0,Y 0.0,Z 0.0,A 0.0,B 0.0,C 0.0}
XYZ_MESS_POS[8,1]={X 0.0,Y 0.0,Z 0.0,A 0.0,B 0.0,C 0.0}
XYZ_MESS_POS[8,2]={X 0.0,Y 0.0,Z 0.0,A 0.0,B 0.0,C 0.0}
XYZ_MESS_POS[8,3]={X 0.0,Y 0.0,Z 0.0,A 0.0,B 0.0,C 0.0}
GLOBAL FRAME XYZ_REF_POS[8,3]
XYZ_REF_POS[1,1]={X 0.0,Y 0.0,Z 0.0,A 0.0,B 0.0,C 0.0}
XYZ_REF_POS[1,2]={X 0.0,Y 0.0,Z 0.0,A 0.0,B 0.0,C 0.0}
XYZ_REF_POS[1,3]={X 0.0,Y 0.0,Z 0.0,A 0.0,B 0.0,C 0.0}
XYZ_REF_POS[2,1]={X 0.0,Y 0.0,Z 0.0,A 0.0,B 0.0,C 0.0}
XYZ_REF_POS[2,2]={X 0.0,Y 0.0,Z 0.0,A 0.0,B 0.0,C 0.0}
XYZ_REF_POS[2,3]={X 0.0,Y 0.0,Z 0.0,A 0.0,B 0.0,C 0.0}
XYZ_REF_POS[3,1]={X 0.0,Y 0.0,Z 0.0,A 0.0,B 0.0,C 0.0}
XYZ_REF_POS[3,2]={X 0.0,Y 0.0,Z 0.0,A 0.0,B 0.0,C 0.0}
XYZ_REF_POS[3,3]={X 0.0,Y 0.0,Z 0.0,A 0.0,B 0.0,C 0.0}
XYZ_REF_POS[4,1]={X 0.0,Y 0.0,Z 0.0,A 0.0,B 0.0,C 0.0}
XYZ_REF_POS[4,2]={X 0.0,Y 0.0,Z 0.0,A 0.0,B 0.0,C 0.0}
XYZ_REF_POS[4,3]={X 0.0,Y 0.0,Z 0.0,A 0.0,B 0.0,C 0.0}
XYZ_REF_POS[5,1]={X 0.0,Y 0.0,Z 0.0,A 0.0,B 0.0,C 0.0}
XYZ_REF_POS[5,2]={X 0.0,Y 0.0,Z 0.0,A 0.0,B 0.0,C 0.0}
XYZ_REF_POS[5,3]={X 0.0,Y 0.0,Z 0.0,A 0.0,B 0.0,C 0.0}
XYZ_REF_POS[6,1]={X 0.0,Y 0.0,Z 0.0,A 0.0,B 0.0,C 0.0}
XYZ_REF_POS[6,2]={X 0.0,Y 0.0,Z 0.0,A 0.0,B 0.0,C 0.0}
XYZ_REF_POS[6,3]={X 0.0,Y 0.0,Z 0.0,A 0.0,B 0.0,C 0.0}
XYZ_REF_POS[7,1]={X 0.0,Y 0.0,Z 0.0,A 0.0,B 0.0,C 0.0}
XYZ_REF_POS[7,2]={X 0.0,Y 0.0,Z 0.0,A 0.0,B 0.0,C 0.0}
XYZ_REF_POS[7,3]={X 0.0,Y 0.0,Z 0.0,A 0.0,B 0.0,C 0.0}
XYZ_REF_POS[8,1]={X 0.0,Y 0.0,Z 0.0,A 0.0,B 0.0,C 0.0}
XYZ_REF_POS[8,2]={X 0.0,Y 0.0,Z 0.0,A 0.0,B 0.0,C 0.0}
XYZ_REF_POS[8,3]={X 0.0,Y 0.0,Z 0.0,A 0.0,B 0.0,C 0.0}
;ENDFOLD FRAMES
;
;FOLD OTHERS
DECL DATE DATUM
STRUC KORR_NEU CHAR KORR_WERT[50],CHAR KORR_DATUM[20]
DECL KORR_NEU KORR_TAB[50]
KORR_TAB[1]={KORR_WERT[] "                                                ",KORR_DATUM[] "                    "}
KORR_TAB[2]={KORR_WERT[] "                                                ",KORR_DATUM[] "                    "}
KORR_TAB[3]={KORR_WERT[] "                                                ",KORR_DATUM[] "                    "}
KORR_TAB[4]={KORR_WERT[] "                                                ",KORR_DATUM[] "                    "}
KORR_TAB[5]={KORR_WERT[] "                                                ",KORR_DATUM[] "                    "}
KORR_TAB[6]={KORR_WERT[] "                                                ",KORR_DATUM[] "                    "}
KORR_TAB[7]={KORR_WERT[] "                                                ",KORR_DATUM[] "                    "}
KORR_TAB[8]={KORR_WERT[] "                                                ",KORR_DATUM[] "                    "}
KORR_TAB[9]={KORR_WERT[] "                                                ",KORR_DATUM[] "                    "}
KORR_TAB[10]={KORR_WERT[] "                                                ",KORR_DATUM[] "                    "}
KORR_TAB[11]={KORR_WERT[] "                                                ",KORR_DATUM[] "                    "}
KORR_TAB[12]={KORR_WERT[] "                                                ",KORR_DATUM[] "                    "}
KORR_TAB[13]={KORR_WERT[] "                                                ",KORR_DATUM[] "                    "}
KORR_TAB[14]={KORR_WERT[] "                                                ",KORR_DATUM[] "                    "}
KORR_TAB[15]={KORR_WERT[] "                                                ",KORR_DATUM[] "                    "}
KORR_TAB[16]={KORR_WERT[] "                                                ",KORR_DATUM[] "                    "}
KORR_TAB[17]={KORR_WERT[] "                                                ",KORR_DATUM[] "                    "}
KORR_TAB[18]={KORR_WERT[] "                                                ",KORR_DATUM[] "                    "}
KORR_TAB[19]={KORR_WERT[] "                                                ",KORR_DATUM[] "                    "}
KORR_TAB[20]={KORR_WERT[] "                                                ",KORR_DATUM[] "                    "}
KORR_TAB[21]={KORR_WERT[] "                                                ",KORR_DATUM[] "                    "}
KORR_TAB[22]={KORR_WERT[] "                                                ",KORR_DATUM[] "                    "}
KORR_TAB[23]={KORR_WERT[] "                                                ",KORR_DATUM[] "                    "}
KORR_TAB[24]={KORR_WERT[] "                                                ",KORR_DATUM[] "                    "}
KORR_TAB[25]={KORR_WERT[] "                                                ",KORR_DATUM[] "                    "}
KORR_TAB[26]={KORR_WERT[] "                                                ",KORR_DATUM[] "                    "}
KORR_TAB[27]={KORR_WERT[] "                                                ",KORR_DATUM[] "                    "}
KORR_TAB[28]={KORR_WERT[] "                                                ",KORR_DATUM[] "                    "}
KORR_TAB[29]={KORR_WERT[] "                                                ",KORR_DATUM[] "                    "}
KORR_TAB[30]={KORR_WERT[] "                                                ",KORR_DATUM[] "                    "}
KORR_TAB[31]={KORR_WERT[] "                                                ",KORR_DATUM[] "                    "}
KORR_TAB[32]={KORR_WERT[] "                                                ",KORR_DATUM[] "                    "}
KORR_TAB[33]={KORR_WERT[] "                                                ",KORR_DATUM[] "                    "}
KORR_TAB[34]={KORR_WERT[] "                                                ",KORR_DATUM[] "                    "}
KORR_TAB[35]={KORR_WERT[] "                                                ",KORR_DATUM[] "                    "}
KORR_TAB[36]={KORR_WERT[] "                                                ",KORR_DATUM[] "                    "}
KORR_TAB[37]={KORR_WERT[] "                                                ",KORR_DATUM[] "                    "}
KORR_TAB[38]={KORR_WERT[] "                                                ",KORR_DATUM[] "                    "}
KORR_TAB[39]={KORR_WERT[] "                                                ",KORR_DATUM[] "                    "}
KORR_TAB[40]={KORR_WERT[] "                                                ",KORR_DATUM[] "                    "}
KORR_TAB[41]={KORR_WERT[] "                                                ",KORR_DATUM[] "                    "}
KORR_TAB[42]={KORR_WERT[] "                                                ",KORR_DATUM[] "                    "}
KORR_TAB[43]={KORR_WERT[] "                                                ",KORR_DATUM[] "                    "}
KORR_TAB[44]={KORR_WERT[] "                                                ",KORR_DATUM[] "                    "}
KORR_TAB[45]={KORR_WERT[] "                                                ",KORR_DATUM[] "                    "}
KORR_TAB[46]={KORR_WERT[] "                                                ",KORR_DATUM[] "                    "}
KORR_TAB[47]={KORR_WERT[] "                                                ",KORR_DATUM[] "                    "}
KORR_TAB[48]={KORR_WERT[] "                                                ",KORR_DATUM[] "                    "}
KORR_TAB[49]={KORR_WERT[] "                                                ",KORR_DATUM[] "                    "}
KORR_TAB[50]={KORR_WERT[] "                                                ",KORR_DATUM[] "                    "}
;ENDFOLD OTHERS
;
;ENDFOLD (VW_xyz-Scan)
;
;FOLD DZ
;
;FOLD Corrframes
GLOBAL INT logNr=1
GLOBAL INT offset=0
STRUC dz_corrFrames CHAR dzSender[16],CHAR dzCorrType[3],CHAR dzCorr[60],CHAR dzCorrBase[2],CHAR dzLogDatum[20]
DECL dz_corrFrames dzCorrTab[200]
dzCorrTab[1]={dzSender[] "                ",dzCorrType[] "  ",dzCorr[] "                                                  ",dzCorrBase[] "  ",dzLogDatum[] "                   "}
dzCorrTab[2]={dzSender[] "                ",dzCorrType[] "  ",dzCorr[] "                                                  ",dzCorrBase[] "  ",dzLogDatum[] "                   "}
dzCorrTab[3]={dzSender[] "                ",dzCorrType[] "  ",dzCorr[] "                                                  ",dzCorrBase[] "  ",dzLogDatum[] "                   "}
dzCorrTab[4]={dzSender[] "                ",dzCorrType[] "  ",dzCorr[] "                                                  ",dzCorrBase[] "  ",dzLogDatum[] "                   "}
dzCorrTab[5]={dzSender[] "                ",dzCorrType[] "  ",dzCorr[] "                                                  ",dzCorrBase[] "  ",dzLogDatum[] "                   "}
dzCorrTab[6]={dzSender[] "                ",dzCorrType[] "  ",dzCorr[] "                                                  ",dzCorrBase[] "  ",dzLogDatum[] "                   "}
dzCorrTab[7]={dzSender[] "                ",dzCorrType[] "  ",dzCorr[] "                                                  ",dzCorrBase[] "  ",dzLogDatum[] "                   "}
dzCorrTab[8]={dzSender[] "                ",dzCorrType[] "  ",dzCorr[] "                                                  ",dzCorrBase[] "  ",dzLogDatum[] "                   "}
dzCorrTab[9]={dzSender[] "                ",dzCorrType[] "  ",dzCorr[] "                                                  ",dzCorrBase[] "  ",dzLogDatum[] "                   "}
dzCorrTab[10]={dzSender[] "                ",dzCorrType[] "  ",dzCorr[] "                                                  ",dzCorrBase[] "  ",dzLogDatum[] "                   "}
dzCorrTab[11]={dzSender[] "                ",dzCorrType[] "  ",dzCorr[] "                                                  ",dzCorrBase[] "  ",dzLogDatum[] "                   "}
dzCorrTab[12]={dzSender[] "                ",dzCorrType[] "  ",dzCorr[] "                                                  ",dzCorrBase[] "  ",dzLogDatum[] "                   "}
dzCorrTab[13]={dzSender[] "                ",dzCorrType[] "  ",dzCorr[] "                                                  ",dzCorrBase[] "  ",dzLogDatum[] "                   "}
dzCorrTab[14]={dzSender[] "                ",dzCorrType[] "  ",dzCorr[] "                                                  ",dzCorrBase[] "  ",dzLogDatum[] "                   "}
dzCorrTab[15]={dzSender[] "                ",dzCorrType[] "  ",dzCorr[] "                                                  ",dzCorrBase[] "  ",dzLogDatum[] "                   "}
dzCorrTab[16]={dzSender[] "                ",dzCorrType[] "  ",dzCorr[] "                                                  ",dzCorrBase[] "  ",dzLogDatum[] "                   "}
dzCorrTab[17]={dzSender[] "                ",dzCorrType[] "  ",dzCorr[] "                                                  ",dzCorrBase[] "  ",dzLogDatum[] "                   "}
dzCorrTab[18]={dzSender[] "                ",dzCorrType[] "  ",dzCorr[] "                                                  ",dzCorrBase[] "  ",dzLogDatum[] "                   "}
dzCorrTab[19]={dzSender[] "                ",dzCorrType[] "  ",dzCorr[] "                                                  ",dzCorrBase[] "  ",dzLogDatum[] "                   "}
dzCorrTab[20]={dzSender[] "                ",dzCorrType[] "  ",dzCorr[] "                                                  ",dzCorrBase[] "  ",dzLogDatum[] "                   "}
dzCorrTab[21]={dzSender[] "                ",dzCorrType[] "  ",dzCorr[] "                                                  ",dzCorrBase[] "  ",dzLogDatum[] "                   "}
dzCorrTab[22]={dzSender[] "                ",dzCorrType[] "  ",dzCorr[] "                                                  ",dzCorrBase[] "  ",dzLogDatum[] "                   "}
dzCorrTab[23]={dzSender[] "                ",dzCorrType[] "  ",dzCorr[] "                                                  ",dzCorrBase[] "  ",dzLogDatum[] "                   "}
dzCorrTab[24]={dzSender[] "                ",dzCorrType[] "  ",dzCorr[] "                                                  ",dzCorrBase[] "  ",dzLogDatum[] "                   "}
dzCorrTab[25]={dzSender[] "                ",dzCorrType[] "  ",dzCorr[] "                                                  ",dzCorrBase[] "  ",dzLogDatum[] "                   "}
dzCorrTab[26]={dzSender[] "                ",dzCorrType[] "  ",dzCorr[] "                                                  ",dzCorrBase[] "  ",dzLogDatum[] "                   "}
dzCorrTab[27]={dzSender[] "                ",dzCorrType[] "  ",dzCorr[] "                                                  ",dzCorrBase[] "  ",dzLogDatum[] "                   "}
dzCorrTab[28]={dzSender[] "                ",dzCorrType[] "  ",dzCorr[] "                                                  ",dzCorrBase[] "  ",dzLogDatum[] "                   "}
dzCorrTab[29]={dzSender[] "                ",dzCorrType[] "  ",dzCorr[] "                                                  ",dzCorrBase[] "  ",dzLogDatum[] "                   "}
dzCorrTab[30]={dzSender[] "                ",dzCorrType[] "  ",dzCorr[] "                                                  ",dzCorrBase[] "  ",dzLogDatum[] "                   "}
dzCorrTab[31]={dzSender[] "                ",dzCorrType[] "  ",dzCorr[] "                                                  ",dzCorrBase[] "  ",dzLogDatum[] "                   "}
dzCorrTab[32]={dzSender[] "                ",dzCorrType[] "  ",dzCorr[] "                                                  ",dzCorrBase[] "  ",dzLogDatum[] "                   "}
dzCorrTab[33]={dzSender[] "                ",dzCorrType[] "  ",dzCorr[] "                                                  ",dzCorrBase[] "  ",dzLogDatum[] "                   "}
dzCorrTab[34]={dzSender[] "                ",dzCorrType[] "  ",dzCorr[] "                                                  ",dzCorrBase[] "  ",dzLogDatum[] "                   "}
dzCorrTab[35]={dzSender[] "                ",dzCorrType[] "  ",dzCorr[] "                                                  ",dzCorrBase[] "  ",dzLogDatum[] "                   "}
dzCorrTab[36]={dzSender[] "                ",dzCorrType[] "  ",dzCorr[] "                                                  ",dzCorrBase[] "  ",dzLogDatum[] "                   "}
dzCorrTab[37]={dzSender[] "                ",dzCorrType[] "  ",dzCorr[] "                                                  ",dzCorrBase[] "  ",dzLogDatum[] "                   "}
dzCorrTab[38]={dzSender[] "                ",dzCorrType[] "  ",dzCorr[] "                                                  ",dzCorrBase[] "  ",dzLogDatum[] "                   "}
dzCorrTab[39]={dzSender[] "                ",dzCorrType[] "  ",dzCorr[] "                                                  ",dzCorrBase[] "  ",dzLogDatum[] "                   "}
dzCorrTab[40]={dzSender[] "                ",dzCorrType[] "  ",dzCorr[] "                                                  ",dzCorrBase[] "  ",dzLogDatum[] "                   "}
dzCorrTab[41]={dzSender[] "                ",dzCorrType[] "  ",dzCorr[] "                                                  ",dzCorrBase[] "  ",dzLogDatum[] "                   "}
dzCorrTab[42]={dzSender[] "                ",dzCorrType[] "  ",dzCorr[] "                                                  ",dzCorrBase[] "  ",dzLogDatum[] "                   "}
dzCorrTab[43]={dzSender[] "                ",dzCorrType[] "  ",dzCorr[] "                                                  ",dzCorrBase[] "  ",dzLogDatum[] "                   "}
dzCorrTab[44]={dzSender[] "                ",dzCorrType[] "  ",dzCorr[] "                                                  ",dzCorrBase[] "  ",dzLogDatum[] "                   "}
dzCorrTab[45]={dzSender[] "                ",dzCorrType[] "  ",dzCorr[] "                                                  ",dzCorrBase[] "  ",dzLogDatum[] "                   "}
dzCorrTab[46]={dzSender[] "                ",dzCorrType[] "  ",dzCorr[] "                                                  ",dzCorrBase[] "  ",dzLogDatum[] "                   "}
dzCorrTab[47]={dzSender[] "                ",dzCorrType[] "  ",dzCorr[] "                                                  ",dzCorrBase[] "  ",dzLogDatum[] "                   "}
dzCorrTab[48]={dzSender[] "                ",dzCorrType[] "  ",dzCorr[] "                                                  ",dzCorrBase[] "  ",dzLogDatum[] "                   "}
dzCorrTab[49]={dzSender[] "                ",dzCorrType[] "  ",dzCorr[] "                                                  ",dzCorrBase[] "  ",dzLogDatum[] "                   "}
dzCorrTab[50]={dzSender[] "                ",dzCorrType[] "  ",dzCorr[] "                                                  ",dzCorrBase[] "  ",dzLogDatum[] "                   "}
dzCorrTab[51]={dzSender[] "                ",dzCorrType[] "  ",dzCorr[] "                                                  ",dzCorrBase[] "  ",dzLogDatum[] "                   "}
dzCorrTab[52]={dzSender[] "                ",dzCorrType[] "  ",dzCorr[] "                                                  ",dzCorrBase[] "  ",dzLogDatum[] "                   "}
dzCorrTab[53]={dzSender[] "                ",dzCorrType[] "  ",dzCorr[] "                                                  ",dzCorrBase[] "  ",dzLogDatum[] "                   "}
dzCorrTab[54]={dzSender[] "                ",dzCorrType[] "  ",dzCorr[] "                                                  ",dzCorrBase[] "  ",dzLogDatum[] "                   "}
dzCorrTab[55]={dzSender[] "                ",dzCorrType[] "  ",dzCorr[] "                                                  ",dzCorrBase[] "  ",dzLogDatum[] "                   "}
dzCorrTab[56]={dzSender[] "                ",dzCorrType[] "  ",dzCorr[] "                                                  ",dzCorrBase[] "  ",dzLogDatum[] "                   "}
dzCorrTab[57]={dzSender[] "                ",dzCorrType[] "  ",dzCorr[] "                                                  ",dzCorrBase[] "  ",dzLogDatum[] "                   "}
dzCorrTab[58]={dzSender[] "                ",dzCorrType[] "  ",dzCorr[] "                                                  ",dzCorrBase[] "  ",dzLogDatum[] "                   "}
dzCorrTab[59]={dzSender[] "                ",dzCorrType[] "  ",dzCorr[] "                                                  ",dzCorrBase[] "  ",dzLogDatum[] "                   "}
dzCorrTab[60]={dzSender[] "                ",dzCorrType[] "  ",dzCorr[] "                                                  ",dzCorrBase[] "  ",dzLogDatum[] "                   "}
dzCorrTab[61]={dzSender[] "                ",dzCorrType[] "  ",dzCorr[] "                                                  ",dzCorrBase[] "  ",dzLogDatum[] "                   "}
dzCorrTab[62]={dzSender[] "                ",dzCorrType[] "  ",dzCorr[] "                                                  ",dzCorrBase[] "  ",dzLogDatum[] "                   "}
dzCorrTab[63]={dzSender[] "                ",dzCorrType[] "  ",dzCorr[] "                                                  ",dzCorrBase[] "  ",dzLogDatum[] "                   "}
dzCorrTab[64]={dzSender[] "                ",dzCorrType[] "  ",dzCorr[] "                                                  ",dzCorrBase[] "  ",dzLogDatum[] "                   "}
dzCorrTab[65]={dzSender[] "                ",dzCorrType[] "  ",dzCorr[] "                                                  ",dzCorrBase[] "  ",dzLogDatum[] "                   "}
dzCorrTab[66]={dzSender[] "                ",dzCorrType[] "  ",dzCorr[] "                                                  ",dzCorrBase[] "  ",dzLogDatum[] "                   "}
dzCorrTab[67]={dzSender[] "                ",dzCorrType[] "  ",dzCorr[] "                                                  ",dzCorrBase[] "  ",dzLogDatum[] "                   "}
dzCorrTab[68]={dzSender[] "                ",dzCorrType[] "  ",dzCorr[] "                                                  ",dzCorrBase[] "  ",dzLogDatum[] "                   "}
dzCorrTab[69]={dzSender[] "                ",dzCorrType[] "  ",dzCorr[] "                                                  ",dzCorrBase[] "  ",dzLogDatum[] "                   "}
dzCorrTab[70]={dzSender[] "                ",dzCorrType[] "  ",dzCorr[] "                                                  ",dzCorrBase[] "  ",dzLogDatum[] "                   "}
dzCorrTab[71]={dzSender[] "                ",dzCorrType[] "  ",dzCorr[] "                                                  ",dzCorrBase[] "  ",dzLogDatum[] "                   "}
dzCorrTab[72]={dzSender[] "                ",dzCorrType[] "  ",dzCorr[] "                                                  ",dzCorrBase[] "  ",dzLogDatum[] "                   "}
dzCorrTab[73]={dzSender[] "                ",dzCorrType[] "  ",dzCorr[] "                                                  ",dzCorrBase[] "  ",dzLogDatum[] "                   "}
dzCorrTab[74]={dzSender[] "                ",dzCorrType[] "  ",dzCorr[] "                                                  ",dzCorrBase[] "  ",dzLogDatum[] "                   "}
dzCorrTab[75]={dzSender[] "                ",dzCorrType[] "  ",dzCorr[] "                                                  ",dzCorrBase[] "  ",dzLogDatum[] "                   "}
dzCorrTab[76]={dzSender[] "                ",dzCorrType[] "  ",dzCorr[] "                                                  ",dzCorrBase[] "  ",dzLogDatum[] "                   "}
dzCorrTab[77]={dzSender[] "                ",dzCorrType[] "  ",dzCorr[] "                                                  ",dzCorrBase[] "  ",dzLogDatum[] "                   "}
dzCorrTab[78]={dzSender[] "                ",dzCorrType[] "  ",dzCorr[] "                                                  ",dzCorrBase[] "  ",dzLogDatum[] "                   "}
dzCorrTab[79]={dzSender[] "                ",dzCorrType[] "  ",dzCorr[] "                                                  ",dzCorrBase[] "  ",dzLogDatum[] "                   "}
dzCorrTab[80]={dzSender[] "                ",dzCorrType[] "  ",dzCorr[] "                                                  ",dzCorrBase[] "  ",dzLogDatum[] "                   "}
dzCorrTab[81]={dzSender[] "                ",dzCorrType[] "  ",dzCorr[] "                                                  ",dzCorrBase[] "  ",dzLogDatum[] "                   "}
dzCorrTab[82]={dzSender[] "                ",dzCorrType[] "  ",dzCorr[] "                                                  ",dzCorrBase[] "  ",dzLogDatum[] "                   "}
dzCorrTab[83]={dzSender[] "                ",dzCorrType[] "  ",dzCorr[] "                                                  ",dzCorrBase[] "  ",dzLogDatum[] "                   "}
dzCorrTab[84]={dzSender[] "                ",dzCorrType[] "  ",dzCorr[] "                                                  ",dzCorrBase[] "  ",dzLogDatum[] "                   "}
dzCorrTab[85]={dzSender[] "                ",dzCorrType[] "  ",dzCorr[] "                                                  ",dzCorrBase[] "  ",dzLogDatum[] "                   "}
dzCorrTab[86]={dzSender[] "                ",dzCorrType[] "  ",dzCorr[] "                                                  ",dzCorrBase[] "  ",dzLogDatum[] "                   "}
dzCorrTab[87]={dzSender[] "                ",dzCorrType[] "  ",dzCorr[] "                                                  ",dzCorrBase[] "  ",dzLogDatum[] "                   "}
dzCorrTab[88]={dzSender[] "                ",dzCorrType[] "  ",dzCorr[] "                                                  ",dzCorrBase[] "  ",dzLogDatum[] "                   "}
dzCorrTab[89]={dzSender[] "                ",dzCorrType[] "  ",dzCorr[] "                                                  ",dzCorrBase[] "  ",dzLogDatum[] "                   "}
dzCorrTab[90]={dzSender[] "                ",dzCorrType[] "  ",dzCorr[] "                                                  ",dzCorrBase[] "  ",dzLogDatum[] "                   "}
dzCorrTab[91]={dzSender[] "                ",dzCorrType[] "  ",dzCorr[] "                                                  ",dzCorrBase[] "  ",dzLogDatum[] "                   "}
dzCorrTab[92]={dzSender[] "                ",dzCorrType[] "  ",dzCorr[] "                                                  ",dzCorrBase[] "  ",dzLogDatum[] "                   "}
dzCorrTab[93]={dzSender[] "                ",dzCorrType[] "  ",dzCorr[] "                                                  ",dzCorrBase[] "  ",dzLogDatum[] "                   "}
dzCorrTab[94]={dzSender[] "                ",dzCorrType[] "  ",dzCorr[] "                                                  ",dzCorrBase[] "  ",dzLogDatum[] "                   "}
dzCorrTab[95]={dzSender[] "                ",dzCorrType[] "  ",dzCorr[] "                                                  ",dzCorrBase[] "  ",dzLogDatum[] "                   "}
dzCorrTab[96]={dzSender[] "                ",dzCorrType[] "  ",dzCorr[] "                                                  ",dzCorrBase[] "  ",dzLogDatum[] "                   "}
dzCorrTab[97]={dzSender[] "                ",dzCorrType[] "  ",dzCorr[] "                                                  ",dzCorrBase[] "  ",dzLogDatum[] "                   "}
dzCorrTab[98]={dzSender[] "                ",dzCorrType[] "  ",dzCorr[] "                                                  ",dzCorrBase[] "  ",dzLogDatum[] "                   "}
dzCorrTab[99]={dzSender[] "                ",dzCorrType[] "  ",dzCorr[] "                                                  ",dzCorrBase[] "  ",dzLogDatum[] "                   "}
dzCorrTab[100]={dzSender[] "                ",dzCorrType[] "  ",dzCorr[] "                                                  ",dzCorrBase[] "  ",dzLogDatum[] "                   "}
dzCorrTab[101]={dzSender[] "                ",dzCorrType[] "  ",dzCorr[] "                                                  ",dzCorrBase[] "  ",dzLogDatum[] "                   "}
dzCorrTab[102]={dzSender[] "                ",dzCorrType[] "  ",dzCorr[] "                                                  ",dzCorrBase[] "  ",dzLogDatum[] "                   "}
dzCorrTab[103]={dzSender[] "                ",dzCorrType[] "  ",dzCorr[] "                                                  ",dzCorrBase[] "  ",dzLogDatum[] "                   "}
dzCorrTab[104]={dzSender[] "                ",dzCorrType[] "  ",dzCorr[] "                                                  ",dzCorrBase[] "  ",dzLogDatum[] "                   "}
dzCorrTab[105]={dzSender[] "                ",dzCorrType[] "  ",dzCorr[] "                                                  ",dzCorrBase[] "  ",dzLogDatum[] "                   "}
dzCorrTab[106]={dzSender[] "                ",dzCorrType[] "  ",dzCorr[] "                                                  ",dzCorrBase[] "  ",dzLogDatum[] "                   "}
dzCorrTab[107]={dzSender[] "                ",dzCorrType[] "  ",dzCorr[] "                                                  ",dzCorrBase[] "  ",dzLogDatum[] "                   "}
dzCorrTab[108]={dzSender[] "                ",dzCorrType[] "  ",dzCorr[] "                                                  ",dzCorrBase[] "  ",dzLogDatum[] "                   "}
dzCorrTab[109]={dzSender[] "                ",dzCorrType[] "  ",dzCorr[] "                                                  ",dzCorrBase[] "  ",dzLogDatum[] "                   "}
dzCorrTab[110]={dzSender[] "                ",dzCorrType[] "  ",dzCorr[] "                                                  ",dzCorrBase[] "  ",dzLogDatum[] "                   "}
dzCorrTab[111]={dzSender[] "                ",dzCorrType[] "  ",dzCorr[] "                                                  ",dzCorrBase[] "  ",dzLogDatum[] "                   "}
dzCorrTab[112]={dzSender[] "                ",dzCorrType[] "  ",dzCorr[] "                                                  ",dzCorrBase[] "  ",dzLogDatum[] "                   "}
dzCorrTab[113]={dzSender[] "                ",dzCorrType[] "  ",dzCorr[] "                                                  ",dzCorrBase[] "  ",dzLogDatum[] "                   "}
dzCorrTab[114]={dzSender[] "                ",dzCorrType[] "  ",dzCorr[] "                                                  ",dzCorrBase[] "  ",dzLogDatum[] "                   "}
dzCorrTab[115]={dzSender[] "                ",dzCorrType[] "  ",dzCorr[] "                                                  ",dzCorrBase[] "  ",dzLogDatum[] "                   "}
dzCorrTab[116]={dzSender[] "                ",dzCorrType[] "  ",dzCorr[] "                                                  ",dzCorrBase[] "  ",dzLogDatum[] "                   "}
dzCorrTab[117]={dzSender[] "                ",dzCorrType[] "  ",dzCorr[] "                                                  ",dzCorrBase[] "  ",dzLogDatum[] "                   "}
dzCorrTab[118]={dzSender[] "                ",dzCorrType[] "  ",dzCorr[] "                                                  ",dzCorrBase[] "  ",dzLogDatum[] "                   "}
dzCorrTab[119]={dzSender[] "                ",dzCorrType[] "  ",dzCorr[] "                                                  ",dzCorrBase[] "  ",dzLogDatum[] "                   "}
dzCorrTab[120]={dzSender[] "                ",dzCorrType[] "  ",dzCorr[] "                                                  ",dzCorrBase[] "  ",dzLogDatum[] "                   "}
dzCorrTab[121]={dzSender[] "                ",dzCorrType[] "  ",dzCorr[] "                                                  ",dzCorrBase[] "  ",dzLogDatum[] "                   "}
dzCorrTab[122]={dzSender[] "                ",dzCorrType[] "  ",dzCorr[] "                                                  ",dzCorrBase[] "  ",dzLogDatum[] "                   "}
dzCorrTab[123]={dzSender[] "                ",dzCorrType[] "  ",dzCorr[] "                                                  ",dzCorrBase[] "  ",dzLogDatum[] "                   "}
dzCorrTab[124]={dzSender[] "                ",dzCorrType[] "  ",dzCorr[] "                                                  ",dzCorrBase[] "  ",dzLogDatum[] "                   "}
dzCorrTab[125]={dzSender[] "                ",dzCorrType[] "  ",dzCorr[] "                                                  ",dzCorrBase[] "  ",dzLogDatum[] "                   "}
dzCorrTab[126]={dzSender[] "                ",dzCorrType[] "  ",dzCorr[] "                                                  ",dzCorrBase[] "  ",dzLogDatum[] "                   "}
dzCorrTab[127]={dzSender[] "                ",dzCorrType[] "  ",dzCorr[] "                                                  ",dzCorrBase[] "  ",dzLogDatum[] "                   "}
dzCorrTab[128]={dzSender[] "                ",dzCorrType[] "  ",dzCorr[] "                                                  ",dzCorrBase[] "  ",dzLogDatum[] "                   "}
dzCorrTab[129]={dzSender[] "                ",dzCorrType[] "  ",dzCorr[] "                                                  ",dzCorrBase[] "  ",dzLogDatum[] "                   "}
dzCorrTab[130]={dzSender[] "                ",dzCorrType[] "  ",dzCorr[] "                                                  ",dzCorrBase[] "  ",dzLogDatum[] "                   "}
dzCorrTab[131]={dzSender[] "                ",dzCorrType[] "  ",dzCorr[] "                                                  ",dzCorrBase[] "  ",dzLogDatum[] "                   "}
dzCorrTab[132]={dzSender[] "                ",dzCorrType[] "  ",dzCorr[] "                                                  ",dzCorrBase[] "  ",dzLogDatum[] "                   "}
dzCorrTab[133]={dzSender[] "                ",dzCorrType[] "  ",dzCorr[] "                                                  ",dzCorrBase[] "  ",dzLogDatum[] "                   "}
dzCorrTab[134]={dzSender[] "                ",dzCorrType[] "  ",dzCorr[] "                                                  ",dzCorrBase[] "  ",dzLogDatum[] "                   "}
dzCorrTab[135]={dzSender[] "                ",dzCorrType[] "  ",dzCorr[] "                                                  ",dzCorrBase[] "  ",dzLogDatum[] "                   "}
dzCorrTab[136]={dzSender[] "                ",dzCorrType[] "  ",dzCorr[] "                                                  ",dzCorrBase[] "  ",dzLogDatum[] "                   "}
dzCorrTab[137]={dzSender[] "                ",dzCorrType[] "  ",dzCorr[] "                                                  ",dzCorrBase[] "  ",dzLogDatum[] "                   "}
dzCorrTab[138]={dzSender[] "                ",dzCorrType[] "  ",dzCorr[] "                                                  ",dzCorrBase[] "  ",dzLogDatum[] "                   "}
dzCorrTab[139]={dzSender[] "                ",dzCorrType[] "  ",dzCorr[] "                                                  ",dzCorrBase[] "  ",dzLogDatum[] "                   "}
dzCorrTab[140]={dzSender[] "                ",dzCorrType[] "  ",dzCorr[] "                                                  ",dzCorrBase[] "  ",dzLogDatum[] "                   "}
dzCorrTab[141]={dzSender[] "                ",dzCorrType[] "  ",dzCorr[] "                                                  ",dzCorrBase[] "  ",dzLogDatum[] "                   "}
dzCorrTab[142]={dzSender[] "                ",dzCorrType[] "  ",dzCorr[] "                                                  ",dzCorrBase[] "  ",dzLogDatum[] "                   "}
dzCorrTab[143]={dzSender[] "                ",dzCorrType[] "  ",dzCorr[] "                                                  ",dzCorrBase[] "  ",dzLogDatum[] "                   "}
dzCorrTab[144]={dzSender[] "                ",dzCorrType[] "  ",dzCorr[] "                                                  ",dzCorrBase[] "  ",dzLogDatum[] "                   "}
dzCorrTab[145]={dzSender[] "                ",dzCorrType[] "  ",dzCorr[] "                                                  ",dzCorrBase[] "  ",dzLogDatum[] "                   "}
dzCorrTab[146]={dzSender[] "                ",dzCorrType[] "  ",dzCorr[] "                                                  ",dzCorrBase[] "  ",dzLogDatum[] "                   "}
dzCorrTab[147]={dzSender[] "                ",dzCorrType[] "  ",dzCorr[] "                                                  ",dzCorrBase[] "  ",dzLogDatum[] "                   "}
dzCorrTab[148]={dzSender[] "                ",dzCorrType[] "  ",dzCorr[] "                                                  ",dzCorrBase[] "  ",dzLogDatum[] "                   "}
dzCorrTab[149]={dzSender[] "                ",dzCorrType[] "  ",dzCorr[] "                                                  ",dzCorrBase[] "  ",dzLogDatum[] "                   "}
dzCorrTab[150]={dzSender[] "                ",dzCorrType[] "  ",dzCorr[] "                                                  ",dzCorrBase[] "  ",dzLogDatum[] "                   "}
dzCorrTab[151]={dzSender[] "                ",dzCorrType[] "  ",dzCorr[] "                                                  ",dzCorrBase[] "  ",dzLogDatum[] "                   "}
dzCorrTab[152]={dzSender[] "                ",dzCorrType[] "  ",dzCorr[] "                                                  ",dzCorrBase[] "  ",dzLogDatum[] "                   "}
dzCorrTab[153]={dzSender[] "                ",dzCorrType[] "  ",dzCorr[] "                                                  ",dzCorrBase[] "  ",dzLogDatum[] "                   "}
dzCorrTab[154]={dzSender[] "                ",dzCorrType[] "  ",dzCorr[] "                                                  ",dzCorrBase[] "  ",dzLogDatum[] "                   "}
dzCorrTab[155]={dzSender[] "                ",dzCorrType[] "  ",dzCorr[] "                                                  ",dzCorrBase[] "  ",dzLogDatum[] "                   "}
dzCorrTab[156]={dzSender[] "                ",dzCorrType[] "  ",dzCorr[] "                                                  ",dzCorrBase[] "  ",dzLogDatum[] "                   "}
dzCorrTab[157]={dzSender[] "                ",dzCorrType[] "  ",dzCorr[] "                                                  ",dzCorrBase[] "  ",dzLogDatum[] "                   "}
dzCorrTab[158]={dzSender[] "                ",dzCorrType[] "  ",dzCorr[] "                                                  ",dzCorrBase[] "  ",dzLogDatum[] "                   "}
dzCorrTab[159]={dzSender[] "                ",dzCorrType[] "  ",dzCorr[] "                                                  ",dzCorrBase[] "  ",dzLogDatum[] "                   "}
dzCorrTab[160]={dzSender[] "                ",dzCorrType[] "  ",dzCorr[] "                                                  ",dzCorrBase[] "  ",dzLogDatum[] "                   "}
dzCorrTab[161]={dzSender[] "                ",dzCorrType[] "  ",dzCorr[] "                                                  ",dzCorrBase[] "  ",dzLogDatum[] "                   "}
dzCorrTab[162]={dzSender[] "                ",dzCorrType[] "  ",dzCorr[] "                                                  ",dzCorrBase[] "  ",dzLogDatum[] "                   "}
dzCorrTab[163]={dzSender[] "                ",dzCorrType[] "  ",dzCorr[] "                                                  ",dzCorrBase[] "  ",dzLogDatum[] "                   "}
dzCorrTab[164]={dzSender[] "                ",dzCorrType[] "  ",dzCorr[] "                                                  ",dzCorrBase[] "  ",dzLogDatum[] "                   "}
dzCorrTab[165]={dzSender[] "                ",dzCorrType[] "  ",dzCorr[] "                                                  ",dzCorrBase[] "  ",dzLogDatum[] "                   "}
dzCorrTab[166]={dzSender[] "                ",dzCorrType[] "  ",dzCorr[] "                                                  ",dzCorrBase[] "  ",dzLogDatum[] "                   "}
dzCorrTab[167]={dzSender[] "                ",dzCorrType[] "  ",dzCorr[] "                                                  ",dzCorrBase[] "  ",dzLogDatum[] "                   "}
dzCorrTab[168]={dzSender[] "                ",dzCorrType[] "  ",dzCorr[] "                                                  ",dzCorrBase[] "  ",dzLogDatum[] "                   "}
dzCorrTab[169]={dzSender[] "                ",dzCorrType[] "  ",dzCorr[] "                                                  ",dzCorrBase[] "  ",dzLogDatum[] "                   "}
dzCorrTab[170]={dzSender[] "                ",dzCorrType[] "  ",dzCorr[] "                                                  ",dzCorrBase[] "  ",dzLogDatum[] "                   "}
dzCorrTab[171]={dzSender[] "                ",dzCorrType[] "  ",dzCorr[] "                                                  ",dzCorrBase[] "  ",dzLogDatum[] "                   "}
dzCorrTab[172]={dzSender[] "                ",dzCorrType[] "  ",dzCorr[] "                                                  ",dzCorrBase[] "  ",dzLogDatum[] "                   "}
dzCorrTab[173]={dzSender[] "                ",dzCorrType[] "  ",dzCorr[] "                                                  ",dzCorrBase[] "  ",dzLogDatum[] "                   "}
dzCorrTab[174]={dzSender[] "                ",dzCorrType[] "  ",dzCorr[] "                                                  ",dzCorrBase[] "  ",dzLogDatum[] "                   "}
dzCorrTab[175]={dzSender[] "                ",dzCorrType[] "  ",dzCorr[] "                                                  ",dzCorrBase[] "  ",dzLogDatum[] "                   "}
dzCorrTab[176]={dzSender[] "                ",dzCorrType[] "  ",dzCorr[] "                                                  ",dzCorrBase[] "  ",dzLogDatum[] "                   "}
dzCorrTab[177]={dzSender[] "                ",dzCorrType[] "  ",dzCorr[] "                                                  ",dzCorrBase[] "  ",dzLogDatum[] "                   "}
dzCorrTab[178]={dzSender[] "                ",dzCorrType[] "  ",dzCorr[] "                                                  ",dzCorrBase[] "  ",dzLogDatum[] "                   "}
dzCorrTab[179]={dzSender[] "                ",dzCorrType[] "  ",dzCorr[] "                                                  ",dzCorrBase[] "  ",dzLogDatum[] "                   "}
dzCorrTab[180]={dzSender[] "                ",dzCorrType[] "  ",dzCorr[] "                                                  ",dzCorrBase[] "  ",dzLogDatum[] "                   "}
dzCorrTab[181]={dzSender[] "                ",dzCorrType[] "  ",dzCorr[] "                                                  ",dzCorrBase[] "  ",dzLogDatum[] "                   "}
dzCorrTab[182]={dzSender[] "                ",dzCorrType[] "  ",dzCorr[] "                                                  ",dzCorrBase[] "  ",dzLogDatum[] "                   "}
dzCorrTab[183]={dzSender[] "                ",dzCorrType[] "  ",dzCorr[] "                                                  ",dzCorrBase[] "  ",dzLogDatum[] "                   "}
dzCorrTab[184]={dzSender[] "                ",dzCorrType[] "  ",dzCorr[] "                                                  ",dzCorrBase[] "  ",dzLogDatum[] "                   "}
dzCorrTab[185]={dzSender[] "                ",dzCorrType[] "  ",dzCorr[] "                                                  ",dzCorrBase[] "  ",dzLogDatum[] "                   "}
dzCorrTab[186]={dzSender[] "                ",dzCorrType[] "  ",dzCorr[] "                                                  ",dzCorrBase[] "  ",dzLogDatum[] "                   "}
dzCorrTab[187]={dzSender[] "                ",dzCorrType[] "  ",dzCorr[] "                                                  ",dzCorrBase[] "  ",dzLogDatum[] "                   "}
dzCorrTab[188]={dzSender[] "                ",dzCorrType[] "  ",dzCorr[] "                                                  ",dzCorrBase[] "  ",dzLogDatum[] "                   "}
dzCorrTab[189]={dzSender[] "                ",dzCorrType[] "  ",dzCorr[] "                                                  ",dzCorrBase[] "  ",dzLogDatum[] "                   "}
dzCorrTab[190]={dzSender[] "                ",dzCorrType[] "  ",dzCorr[] "                                                  ",dzCorrBase[] "  ",dzLogDatum[] "                   "}
dzCorrTab[191]={dzSender[] "                ",dzCorrType[] "  ",dzCorr[] "                                                  ",dzCorrBase[] "  ",dzLogDatum[] "                   "}
dzCorrTab[192]={dzSender[] "                ",dzCorrType[] "  ",dzCorr[] "                                                  ",dzCorrBase[] "  ",dzLogDatum[] "                   "}
dzCorrTab[193]={dzSender[] "                ",dzCorrType[] "  ",dzCorr[] "                                                  ",dzCorrBase[] "  ",dzLogDatum[] "                   "}
dzCorrTab[194]={dzSender[] "                ",dzCorrType[] "  ",dzCorr[] "                                                  ",dzCorrBase[] "  ",dzLogDatum[] "                   "}
dzCorrTab[195]={dzSender[] "                ",dzCorrType[] "  ",dzCorr[] "                                                  ",dzCorrBase[] "  ",dzLogDatum[] "                   "}
dzCorrTab[196]={dzSender[] "                ",dzCorrType[] "  ",dzCorr[] "                                                  ",dzCorrBase[] "  ",dzLogDatum[] "                   "}
dzCorrTab[197]={dzSender[] "                ",dzCorrType[] "  ",dzCorr[] "                                                  ",dzCorrBase[] "  ",dzLogDatum[] "                   "}
dzCorrTab[198]={dzSender[] "                ",dzCorrType[] "  ",dzCorr[] "                                                  ",dzCorrBase[] "  ",dzLogDatum[] "                   "}
dzCorrTab[199]={dzSender[] "                ",dzCorrType[] "  ",dzCorr[] "                                                  ",dzCorrBase[] "  ",dzLogDatum[] "                   "}
dzCorrTab[200]={dzSender[] "                ",dzCorrType[] "  ",dzCorr[] "                                                  ",dzCorrBase[] "  ",dzLogDatum[] "                   "}
;ENDFOLD (Corrframes)
;
;ENDFOLD (DZ)
;
;
;***************************************************
;FOLD Meldungsausgabe
ENUM MOD2R_MsgType StateMsg,QuitMsg,NotifyMsg
;ENDFOLD
;***************************************************
;ENDFOLD (MOD2)
;
;***************************************************
;FOLD MOD3
;
;
;***************************************************
;FOLD Meldungsausgabe
ENUM MOD3R_MsgType StateMsg,QuitMsg,NotifyMsg
;ENDFOLD
;***************************************************
;ENDFOLD (MOD3)
;
;***************************************************
ENDDAT
